FUNCTION_BLOCK Conveyor_HMI
  (* Standard: 61499-2 *)
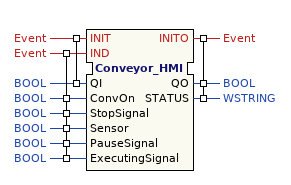
  EVENT_INPUT
    INIT WITH QI;
    IND WITH ConvOn, StopSignal, Sensor, PauseSignal, ExecutingSignal;
  END_EVENT
  EVENT_OUTPUT
    INITO WITH QO, STATUS;
  END_EVENT
  VAR_INPUT
    QI : BOOL;
    ConvOn : BOOL;
    StopSignal : BOOL;
    Sensor : BOOL;
    PauseSignal : BOOL;
    ExecutingSignal : BOOL;
  END_VAR
  VAR_OUTPUT
    QO : BOOL;
    STATUS : WSTRING;
  END_VAR
END_FUNCTION_BLOCK
